{attribute addProperty BoxType "BK1120-0000-0020"}
{attribute addProperty Id "Term_380_KL1002KL1002_D229A9CA00"}
{attribute addProperty CRC "760044134"}
{attribute addProperty SizeInBites "0"}
{attribute addProperty SizeInBytes "0"}
TYPE A_0007_BK1120_0000_0020_2D4D5A66 EXTENDS BK1120_4487A81F :
STRUCT
	{attribute addProperty Name "Term_380_KL1002"}
	Term_380_KL1002 : KL1002_D229A9CA;
END_STRUCT
END_TYPE

(* stored: Version 1.2.0.0, ProductVersion 3.1.4024.9
   DUT A_0007_BK1120_0000_0020_2D4D5A66: Id {9f4796f1-ee00-4243-b5df-6839ae0f7696} *)
